TYPE ST_Sts1_PoseData :
STRUCT
	
	aPoseSmallMotorPickupSt1 : ARRAY [1..6] OF REAL := [-220.552, 67.9 , 150, 180, -20 ,0] ; // Pose before gripper in to the pallet picking position
	aPoseSmallMotorPickupSt2 : ARRAY [1..6] OF REAL := [-220.552, 67.9 , 111.4134, 180, -20 ,0] ;  // Pose before gripper grip, or pose after gripper grip
	aPoseSmallMotorPickupSt3 : ARRAY [1..6] OF REAL := [-222.713, 67.9 , 112.2, 180, -20 ,0] ; //  Pose gripper grip CAN NOT BE MOVEPOSE
	rLinPosSmallMotorPickup				: LREAL := 80; // Linear axis position for pickup functions for selected station
	
	aPoseSmallMotorPlaceSt1 : ARRAY [1..6] OF REAL := [-73.2, 168.6 ,110.6 , 180, 0 ,90] ; // Pose before Small motor in station
	aPoseSmallMotorPlaceSt2 : ARRAY [1..6] OF REAL  := [-73.2, 168.6 ,67.6 , 180, 0 ,90]; // Pose Small motor in station
	rLinPosPlace : LREAL := 10; // Linear axis position for placing functions for selected station

	aPoseMirrorAdj : ARRAY[1..6] OF REAL; // Pose where final position of left mirror is saved in case position adjustment is needed.
	
	aPoseLargeMotorPickupSt1	: ARRAY [1..6] OF REAL := [-124.609, 117.800 , 101.6 , 0, -90 ,0]; // POSE BEFORE ACTUAL GRIP POSITION -108.2
	aPoseLargeMotorPickupSt2	: ARRAY [1..6] OF REAL := [-224.609, 117.800 , 101.6 , 0, -90 ,0];// ACTUAL GRIP POSITION
	aPoseLargeMotorPickupSt3	: ARRAY [1..6] OF REAL := [-224.609, 117.800 , 201.6 , 0, -90 ,0];// MOTOR LIFT FROM PALLET
	rLinPosMotorPickup				: LREAL := 120; // Linear axis position for pickup functions for selected station
	
	aPoseLargeMotorPlaceSt1	: ARRAY [1..6] OF REAL := [-73.3, 80 , 67.6 , 180, 0 ,90]; // POSE BEFORE ACTULA LEAVING POSITION '
	aPoseLargeMotorPlaceSt2	: ARRAY [1..6] OF REAL := [-73.3, 146 , 67.6 , 180, 0 ,90]; // ACTUAL POSITION FOR LEAVING MOTOR AT CURING STATION '
	aPoseLargeMotorPlaceSt3	: ARRAY [1..6] OF REAL := [-73.3, 146 , 100.6 , 180, 0 ,90]; // POSE AFTER LEAVING MOTOR AT CURING STATION '
	
	aPoseMirrorPickupSt1	: ARRAY [1..6] OF REAL := [-158.84, 76.3 , 120, 181, 0 ,0]; // POSE BEFORE ACTUAL GRIP POSITION
	aPoseMirrorPickupSt2	: ARRAY [1..6] OF REAL := [-158.84, 76.3 , 81.55, 181, 0 ,0];// ACTUAL GRIP POSITION 187.1757
	rLinPosMirrorPickup				: LREAL := 80; // Linear axis position for pickup functions for selected station
	
 	aPoseG10MirrorPlaceSt1	: ARRAY [1..6] OF REAL := [-73.3, 190.6 ,117.4 , 180, 0 ,90]; // POSE BEFORE INSERTIN MIRROR IN STATION'
 	aPoseG10MirrorPlaceSt2	: ARRAY [1..6] OF REAL := [-73.3, 188.2 ,70.4 , -180, 0 ,90]; // POSE MIRROR IN STATION BUT NOT INSERTED TO MOTOR '
 	aPoseg10MirrorPlaceSt3	: ARRAY [1..6] OF REAL := [-73.3, 187 ,68.6 , -179, 0 ,90]; // POSE MIRROR INSERTED TO MOTOR'
	
	aPoseG14MirrorPlaceSt1	: ARRAY [1..6] OF REAL := [-73.3, 190.6 ,117.4 , 180, 0 ,90]; // POSE BEFORE INSERTIN MIRROR IN STATION'
	aPoseG14MirrorPlaceSt2	: ARRAY [1..6] OF REAL := [-73.3, 191.6 ,70.4 , -170, 0 ,90]; // POSE MIRROR IN STATION BUT NOT INSERTED TO MOTOR '
	aPoseg14MirrorPlaceSt3	: ARRAY [1..6] OF REAL := [-73.3, 190.1 ,68.6 , -178.5, -0.2 ,90]; // POSE MIRROR INSERTED TO MOTOR'
	
	aPosePassedLargeSt1 		: ARRAY [1..6] OF REAL := [-213.4, 62.25 , 141.45, 180, -20 ,0]; // In and out of pallet
	aPosePassedLargeSt2			: ARRAY [1..6] OF REAL := [-223.4, 62.25 , 101.45, 180, -20 ,0]; // before leaving position
	aPosePassedLargeSt3			: ARRAY [1..6] OF REAL := [-228, 62.25 ,97.79, 180, -20 ,0]; // Leaving position
	
	aPosePassedSmallSt1			: ARRAY [1..6] OF REAL := [-243.3, 42.14 ,157.0, -180, -20 ,0];
	aPosePassedSmallSt2			: ARRAY [1..6] OF REAL := [-243.3, 42.14 ,127.0, -180, -20 ,0];
	aPosePassedSmallSt3			: ARRAY [1..6] OF REAL := [-250.57, 42.14 ,105.640 , -180, -20 ,0];
	
	rLinPosPalletPass : LREAL := 280; // Linear axis position for placing passed assembly for selected station
	rLinPosPalletReject : LREAL; // Linear axis position for placing rejected assembly for selected station
	
END_STRUCT
END_TYPE

(* stored: Version 1.1.0.1
   DUT ST_Sts1_PoseData: Id {00c6b570-8a26-4cce-8861-12d2ac83bc56} *)
